{attribute 'linkalways'} 
{attribute 'no_explicit_call' := 'This FB is a CLASS and must be accessed using methods or properties'}
{attribute 'enable_dynamic_creation'}
FUNCTION_BLOCK KeyValueCollectionChangedEvent EXTENDS KeyValueCollectionEvent IMPLEMENTS I_KeyValueCollectionChangedEvent

END_FUNCTION_BLOCK

(* stored: Version 1.1.0.1, ProductVersion 3.1.4024.12
   POU KeyValueCollectionChangedEvent: Id {64370b37-0020-4f47-bb3e-34b3d8cec17a}, SpecialFunc None *)
